(* LS Electric XG5000 project: COUNTER *)
(* PLC LSPLC *)

FUNCTION_BLOCK water_beam
VAR_INPUT
    sensor : BOOL;
    timer1 : TIME;
    timer2 : TIME;
    timer3 : TIME;
END_VAR
VAR_OUTPUT
    water : BOOL;
END_VAR
VAR
    off1 : TP;
    off2 : TP;
    on1 : TON;
END_VAR

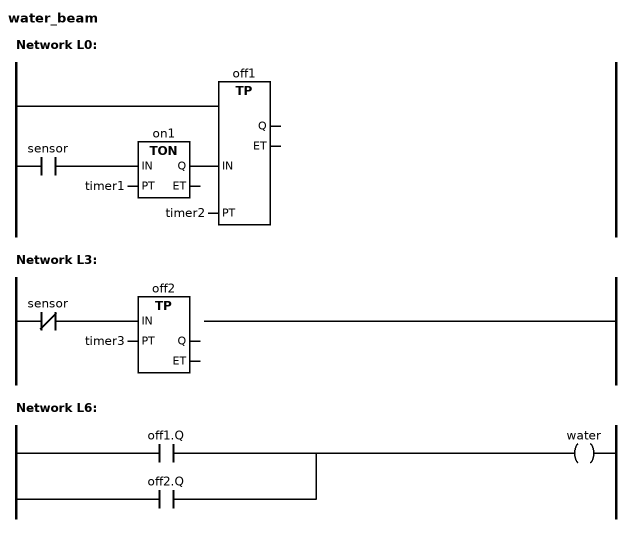
(* Rung L0 *)
on1(IN := sensor, PT := timer1);
off1(IN := on1.Q, PT := timer2);
(* Rung L3 *)
off2(IN := NOT sensor, PT := timer3);
(* Rung L6 *)
water := off1.Q OR off2.Q;
END_FUNCTION_BLOCK

FUNCTION 시간검출 : ARRAY[0..5] OF WORD
VAR_INPUT
    _RTC_TIME_O : BYTE;
    _RTC_TIME_1 : BYTE;
    _RTC_TIME_2 : BYTE;
    _RTC_TIME_3 : BYTE;
    _RTC_TIME_4 : BYTE;
    _RTC_TIME_5 : BYTE;
END_VAR

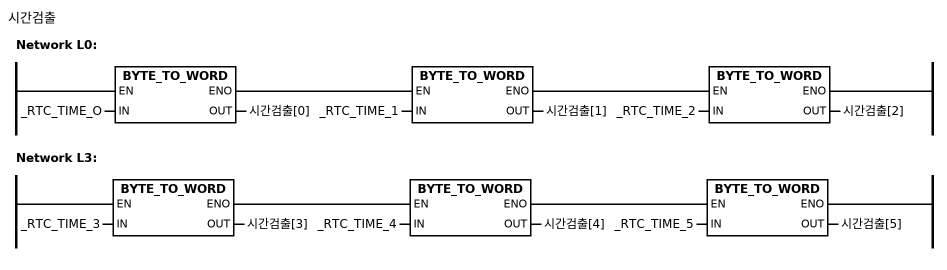
(* Rung L0 *)
시간검출[0] := BYTE_TO_WORD(_RTC_TIME_O);
시간검출[1] := BYTE_TO_WORD(_RTC_TIME_1);
시간검출[2] := BYTE_TO_WORD(_RTC_TIME_2);
(* Rung L3 *)
시간검출[3] := BYTE_TO_WORD(_RTC_TIME_3);
시간검출[4] := BYTE_TO_WORD(_RTC_TIME_4);
시간검출[5] := BYTE_TO_WORD(_RTC_TIME_5);
END_FUNCTION

FUNCTION_BLOCK 사칙연산
VAR_INPUT
    IN1 : REAL;
    IN2 : REAL;
    RESET : BOOL;
END_VAR
VAR_OUTPUT
    ADD_OUT : REAL;
    SUB_OUT : REAL;
    MUL_OUT : REAL;
    DIV_OUT : REAL;
END_VAR

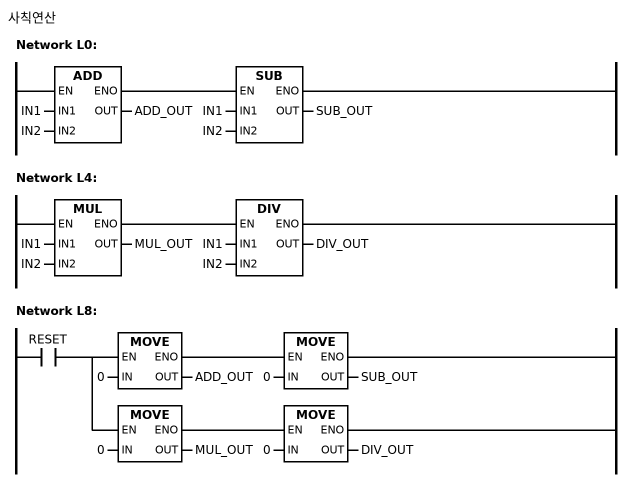
(* Rung L0 *)
ADD_OUT := IN1 + IN2;
SUB_OUT := IN1 - IN2;
(* Rung L4 *)
MUL_OUT := IN1 * IN2;
DIV_OUT := IN1 / IN2;
(* Rung L8 *)
IF RESET THEN
    ADD_OUT := 0;
    SUB_OUT := 0;
    MUL_OUT := 0;
    DIV_OUT := 0;
END_IF;
END_FUNCTION_BLOCK

FUNCTION_BLOCK PITA
VAR_IN_OUT
    B변 : REAL;
    A변 : REAL;
    각A : REAL;
    각B : REAL;
END_VAR
VAR_INPUT
    RESET : BOOL;
END_VAR
VAR_OUTPUT
    Result : REAL;
END_VAR
VAR
    ADD_OUT : REAL;
    A변_제곱 : REAL;
    B변_제곱 : REAL;
    DIV_A : REAL;
    DIV_B : REAL;
    각도환산 : REAL := 57.2957795131;
    라디안A : REAL;
    라디안B : REAL;
END_VAR

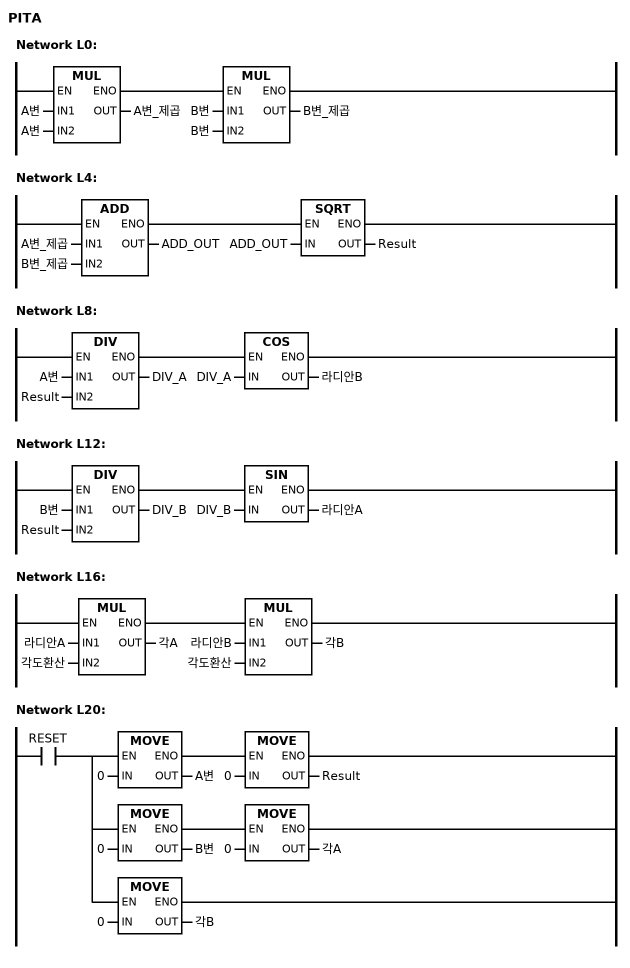
(* Rung L0 *)
A변_제곱 := A변 * A변;
B변_제곱 := B변 * B변;
(* Rung L4 *)
ADD_OUT := A변_제곱 + B변_제곱;
Result := SQRT(ADD_OUT);
(* Rung L8 *)
DIV_A := A변 / Result;
라디안B := COS(DIV_A);
(* Rung L12 *)
DIV_B := B변 / Result;
라디안A := SIN(DIV_B);
(* Rung L16 *)
각A := 라디안A * 각도환산;
각B := 라디안B * 각도환산;
(* Rung L20 *)
IF RESET THEN
    A변 := 0;
    Result := 0;
    B변 := 0;
    각A := 0;
    각B := 0;
END_IF;
END_FUNCTION_BLOCK

FUNCTION_BLOCK 실습2
VAR_INPUT
    FL : BOOL;
    NFL : BOOL;
    OFF : BOOL;
END_VAR
VAR_OUTPUT
    LA1 : BOOL;
    LA2 : BOOL;
END_VAR
VAR
    FLAG : BOOL;
    FUN1 : TP;
END_VAR
VAR
    _e1 : R_TRIG;
    _e2 : R_TRIG;
    _e3 : R_TRIG;
END_VAR

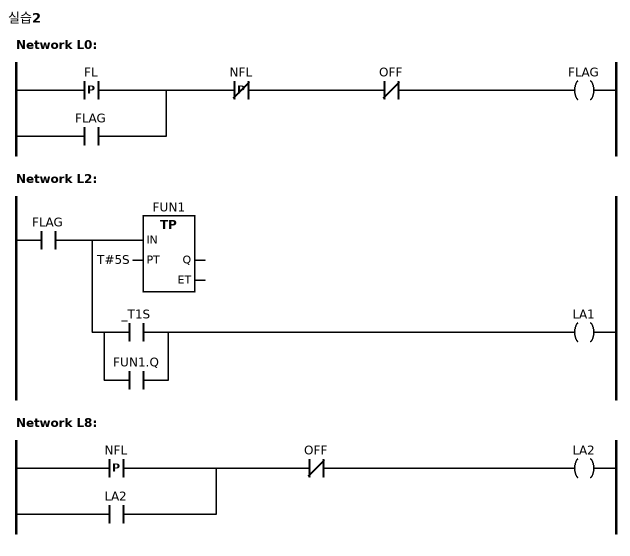
(* Rung L0 *)
_e1(CLK := FL);
_e2(CLK := NFL);
FLAG := (_e1.Q OR FLAG) AND NOT _e2.Q AND NOT OFF;
(* Rung L2 *)
FUN1(IN := FLAG, PT := T#5S);
LA1 := FLAG AND (_T1S OR FUN1.Q);
(* Rung L8 *)
_e3(CLK := NFL);
LA2 := (_e3.Q OR LA2) AND NOT OFF;
END_FUNCTION_BLOCK

PROGRAM NewProgram (* task: 스캔 프로그램 *)
VAR
    A : REAL;
    A2 : REAL;
    B : REAL;
    B2 : REAL;
    BB : BYTE;
    CALC : 사칙연산;
    DEG_A2 : REAL;
    DEG_B2 : REAL;
    exp_in : BOOL;
    exp_out : BOOL;
    FL : BOOL;
    FL_FUN : TON;
    FL_FUN1 : TON;
    FL_FUN1_사본1 : TP;
    FL_FUN2 : TOF;
    INST : CTU_INT;
    INST1 : CTD_INT;
    INST2 : CTUD_DINT;
    INST3 : water_beam;
    INST4 : 사칙연산;
    LA1 : BOOL;
    LA2 : BOOL;
    MONTH : BOOL;
    NFL : BOOL;
    OFF : BOOL;
    ON1 : BOOL;
    ON2 : BOOL;
    OO : WORD;
    OUT : BOOL;
    PRACTICE2 : 실습2;
    Result : REAL;
    sensor : BOOL;
    STOP : BOOL;
    TRIG : BOOL;
    water : BOOL;
    X0 : BOOL;
    X1 : BOOL;
    X2 : BOOL;
    X3 : BOOL;
    X4 : BOOL;
    X5 : BOOL;
    X6 : BOOL;
    X7 : BOOL;
    Y0 : BOOL;
    Y1 : BOOL;
    Y2 : BOOL;
    YEAR : BOOL;
    년 : WORD;
    램프1 : BOOL;
    램프2 : BOOL;
    리셋 : BOOL;
    리셋2 : BOOL;
    분 : WORD;
    사칙연산 : BOOL;
    시 : WORD;
    시간검출 : ARRAY[0..5] OF WORD;
    월 : WORD;
    일 : WORD;
    초 : WORD;
    출력 : BOOL;
    트리거 : BOOL;
    트리거2 : BOOL;
    트리거3 : BOOL;
    트리거4 : BOOL;
    피타고라스 : PITA;
END_VAR
VAR
    _e1 : R_TRIG;
    _e2 : R_TRIG;
    _e3 : R_TRIG;
END_VAR

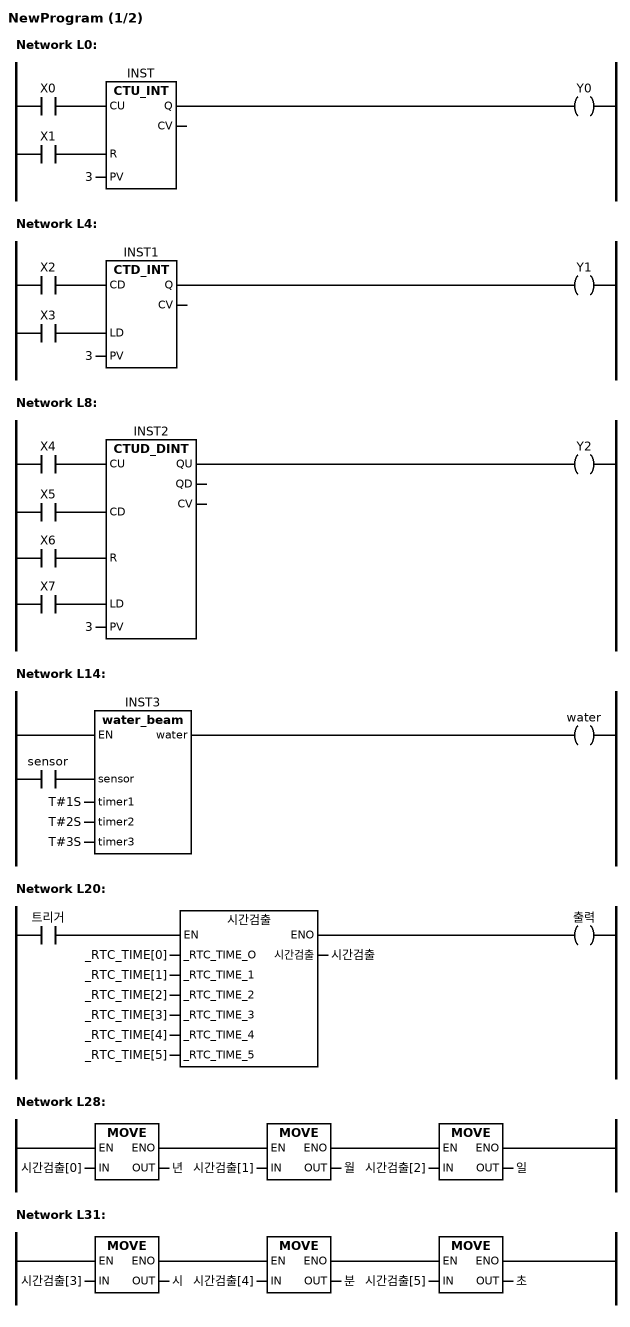
(* Rung L0 *)
INST(CU := X0, R := X1, PV := 3);
Y0 := INST.Q;
(* Rung L4 *)
INST1(CD := X2, LD := X3, PV := 3);
Y1 := INST1.Q;
(* Rung L8 *)
INST2(CU := X4, CD := X5, R := X6, LD := X7, PV := 3);
Y2 := INST2.QU;
(* Rung L14 *)
INST3(sensor := sensor, timer1 := T#1S, timer2 := T#2S, timer3 := T#3S);
water := INST3.water;
(* Rung L20 *)
IF 트리거 THEN
    시간검출 := 시간검출(_RTC_TIME_O := _RTC_TIME[0], _RTC_TIME_1 := _RTC_TIME[1], _RTC_TIME_2 := _RTC_TIME[2], _RTC_TIME_3 := _RTC_TIME[3], _RTC_TIME_4 := _RTC_TIME[4], _RTC_TIME_5 := _RTC_TIME[5]);
END_IF;
출력 := 트리거;
(* Rung L28 *)
년 := 시간검출[0];
월 := 시간검출[1];
일 := 시간검출[2];
(* Rung L31 *)
시 := 시간검출[3];
분 := 시간검출[4];
초 := 시간검출[5];

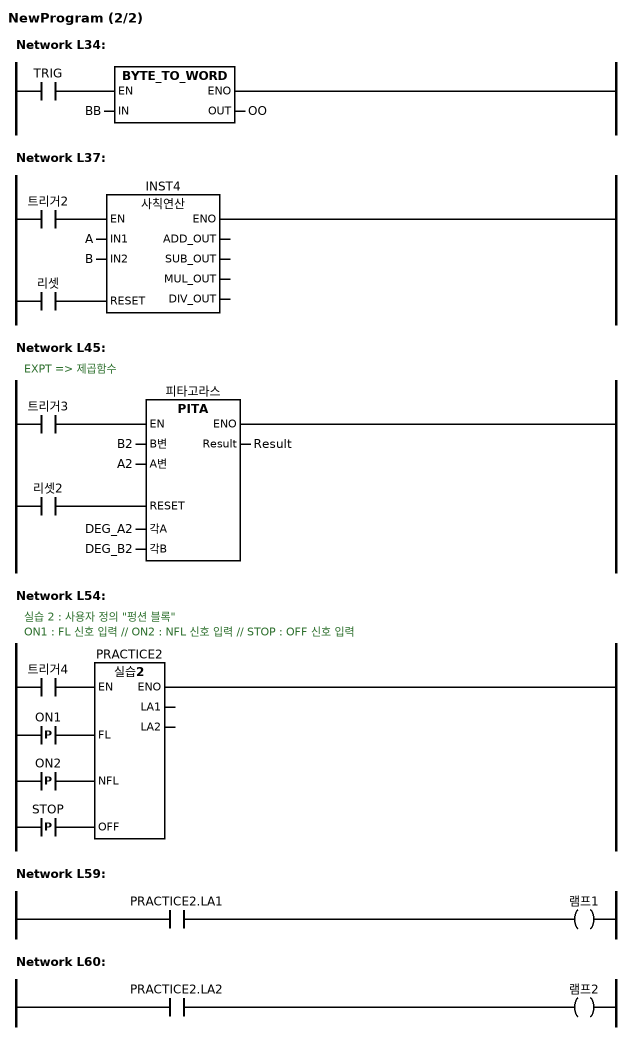
(* Rung L34 *)
IF TRIG THEN OO := BYTE_TO_WORD(BB); END_IF;
(* Rung L37 *)
IF 트리거2 THEN INST4(IN1 := A, IN2 := B, RESET := 리셋); END_IF;
(* EXPT => 제곱함수 *)
(* Rung L45 *)
IF 트리거3 THEN
    피타고라스(B변 := B2, A변 := A2, RESET := 리셋2, 각A := DEG_A2, 각B := DEG_B2, Result => Result);
END_IF;
(* 실습 2 : 사용자 정의 "펑션 블록" *)
(* ON1 : FL 신호 입력 // ON2 : NFL 신호 입력 // STOP : OFF 신호 입력 *)
(* Rung L54 *)
_e1(CLK := ON1);
_e2(CLK := ON2);
_e3(CLK := STOP);
IF 트리거4 THEN PRACTICE2(FL := _e1.Q, NFL := _e2.Q, OFF := _e3.Q); END_IF;
(* Rung L59 *)
램프1 := PRACTICE2.LA1;
(* Rung L60 *)
램프2 := PRACTICE2.LA2;
END_PROGRAM